{attribute 'GeneratedUsingTerminal: EP9128-0020-0016'}
{attribute addProperty BoxType "EP9128-0020-0016"}
{attribute addProperty Id "A_0004_EP9128_0021_0016A_0004_EP9128_0021_0016_EBEEF4C1589A_0001_EP9128_0020_0016_2_EP9128_1020EP9128_1FC0878B2A_0001_EP9128_0020_0016_3_EP9128_2020EP9128_1FC0878B2"}
{attribute addProperty CRC "4026962164"}
{attribute addProperty Size "593"}
TYPE A_0001_EP9128_0020_0016_F00690F4 EXTENDS EP9128_1FC0878B :
STRUCT
	{attribute addProperty Name "A_0004(EP9128-0021-0016)"}
	{attribute addProperty PreviousPort "A_0001(EP9128-0020-0016) : D"}
	A_0004_EP9128_0021_0016 : A_0004_EP9128_0021_0016_EBEEF4C1;
	{attribute addProperty Name "A_0001(EP9128-0020-0016)_2 (EP9128-1020)"}
	{attribute addProperty PreviousPort "A_0001(EP9128-0020-0016) : C"}
	A_0001_EP9128_0020_0016_2_EP9128_1020 : EP9128_1FC0878B;
	{attribute addProperty Name "A_0001(EP9128-0020-0016)_3 (EP9128-2020)"}
	{attribute addProperty PreviousPort "A_0001(EP9128-0020-0016)_2 (EP9128-1020) : C"}
	A_0001_EP9128_0020_0016_3_EP9128_2020 : EP9128_1FC0878B;
END_STRUCT
END_TYPE

(* stored: Version 1.2.0.0, ProductVersion 3.1.4024.9
   DUT A_0001_EP9128_0020_0016_F00690F4: Id {53ca3e5d-8ced-49f9-9ce8-9325e89726fd} *)
